TYPE MidiSmokeParameters :
STRUCT
	{attribute 'TcEncoding':='UTF-8'}
	ModbusTCP_IP: STRING := '192.168.1.234';
END_STRUCT
END_TYPE

(* stored: Version 1.1.0.1, ProductVersion 3.1.4024.6
   DUT MidiSmokeParameters: Id {7fb3c9cf-cff1-4207-a5e7-76686113dc74} *)
